# EPICS autosave request: iocBoot/ioc13bmd_lightfield1/auto_settings.req
file "LightField_settings.req",   P=$(P),  R=cam1:
file "NDStdArrays_settings.req",  P=$(P),  R=image1:
file "commonPlugin_settings.req", P=$(P)
